(* CODESYS project reflex1.project

Project tree, tasks and I/O mapping:
  Device : CODESYS Control Win V3, 3S - Smart Software Solutions GmbH, order no. 305021, version 3.5.8.10
    application Application
      libraries: Standard, * (System); BASIC, 3.31 (OSCAT)
      task MainTask (cyclic, interval t#20ms, priority 1) calls PLC_PRG
      program PLC_PRG [ST]
      visualisation Visualization
  libraries: VisuSymbols, 3.5.8.0 (System)
  text list GlobalTextList
*)

// Device/Application/PLC_PRG
PROGRAM PLC_PRG
VAR
	controls: ARRAY [1..4] OF BOOL;	
	push: ARRAY [1..4] OF BOOL;	

	set: ARRAY [1..15] OF INT;
	set2: ARRAY [1..15] OF INT;
	
	
	index: INT;
	
	t1: TON;
	t2: TOF;
	
	newGame: BOOL := TRUE;
	newGame2: BOOL;
	newGame3: BOOL;
	start: BOOL;
END_VAR

t1(IN:=newGame,PT:=T#1MS);
newGame2 := t1.Q;

IF(newGame2 := TRUE) THEN
	set[1] := RDM2(last:=set[1],low:=1,high:=4);
	newGame3:=FALSE;
END_IF

t2(IN:=newGame3,PT:=T#1MS);
newGame2 := t1.Q;
t2(IN:=newGame2,PT:=T#1MS);
newGame := t1.Q;

IF(set[1] = 1) THEN
	t1(IN:=start,PT:=T#0.1MS);
	controls[1] := t1.Q;
END_IF

IF(set[1] = 2) THEN
	t1(IN:=controls[2],PT:=T#0.1MS);
	controls[2] := t1.Q;
END_IF

IF(set[1] = 3) THEN
	t1(IN:=controls[3],PT:=T#0.1MS);
	controls[3] := t1.Q;
END_IF

IF(set[1] = 4) THEN
	t1(IN:=controls[4],PT:=T#0.1MS);
	controls[4] := t1.Q;
END_IF

END_PROGRAM

// Device/Application/Visualization
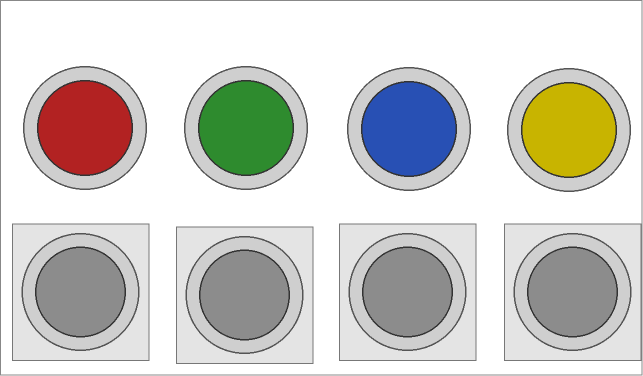
VISUALIZATION Visualization  // 643x376
    Lamp1 (13,39 144x178), variable: PLC_PRG.controls[1], style: Lamp-Lamp1-Red
    Lamp1 (174,39 144x178), variable: PLC_PRG.controls[2], style: Lamp-Lamp1-Green
    Lamp1 (337,40 144x178), variable: PLC_PRG.controls[3], style: Lamp-Lamp1-Blue
    Lamp1 (497,41 144x178), variable: PLC_PRG.controls[4], style: Lamp-Lamp1-Yellow
    PushSwitch (12,213 137x158), variable: PLC_PRG.push[1], behaviour: TOGGLE, style: Switch-PushSwitch-Gray
    PushSwitch (176,216 137x158), variable: PLC_PRG.push[2], behaviour: TOGGLE, style: Switch-PushSwitch-Gray
    PushSwitch (339,213 137x158), variable: PLC_PRG.push[3], behaviour: TOGGLE, style: Switch-PushSwitch-Gray
    PushSwitch (504,213 137x158), variable: PLC_PRG.push[4], behaviour: TOGGLE, style: Switch-PushSwitch-Gray
END_VISUALIZATION
